// TIA Portal V20 export
// export: Created 2025-12-01T14:56:22.3748752Z, ExportSetting None, DisplayName Totally Integrated Automation Portal, DisplayVersion V20 Update 3, DisplayName TIA Portal Openness, DisplayVersion V20 Update 3, DisplayName TIA Portal Version Control Interface, DisplayVersion V20 Update 3, DisplayName STEP 7 Professional, DisplayVersion V20 Update 3, DisplayName STEP 7 Safety, DisplayVersion V20 Update 2, DisplayName WinCC Basic/Comfort/Advanced, DisplayVersion V20 Update 3, DisplayName WinCC Professional, DisplayVersion V20 Update 3, DisplayName WinCC Unified, DisplayVersion V20 Update 3
TYPE "UDT_Elevador_Config"
   STRUCT
      Posicion_mm_H1 : Real;
      Posicion_mm_H2 : Real;
      Derecha : Bool;
      Izquierda : Bool;
   END_STRUCT;
END_TYPE
